TYPE Timer :
STRUCT
	RotateDisc : TON;
	LinearFW : TON;
	GripperLower : TON;
	GripperOpen : TON;
	GripperClose: TON;
	GripperLift: TON;
	LinearBW : TON;
END_STRUCT
END_TYPE

(* stored: Version 1.1.0.1, ProductVersion 3.1.4024.12
   DUT Timer: Id {4f3d270c-4705-44ab-9d69-90aa46096bbf} *)
